Staubli VAL3: GeometryRS.dtx

public num nSyncDist = 1
public num nWinDownStream
public num nWinUpStream
public bool bIsScara
public bool bLinear
public bool bUseUserCenter
public bool bUseUserLimit = true
pointRs pVision[3]
  [0] = {fatherId=world[0]}
  [1] = {fatherId=world[0]}
  [2] = {fatherId=world[0]}
pointRs pWinCenter = {fatherId=world[0]}
pointRs pWinDown[2]
  [0] = {fatherId=world[0]}
  [1] = {fatherId=world[0]}
pointRs pWinMiddle = {fatherId=world[0]}
pointRs pWinUp[2]
  [0] = {fatherId=world[0]}
  [1] = {fatherId=world[0]}
tool pointer = {z=100, fatherId=flange[0], ioLink=valve1}
